Universal Robots URScript: Main Program plate.script

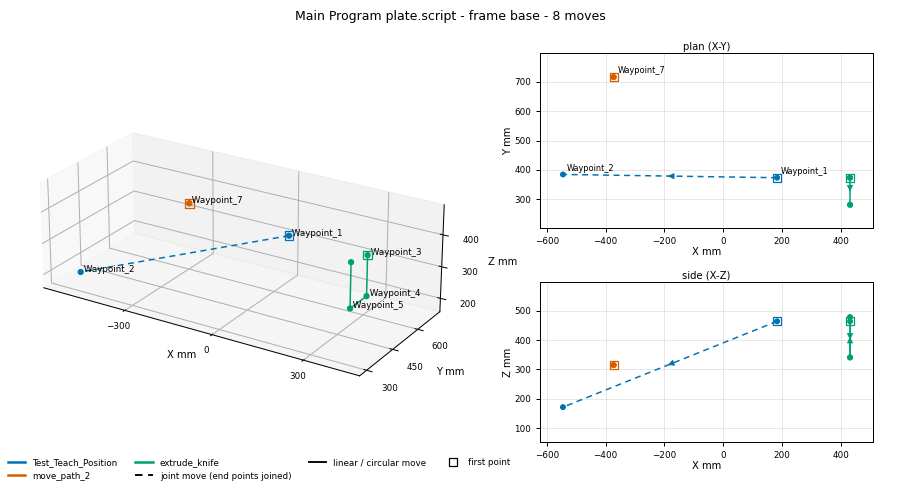
[picture p0: tool path of Main Program plate.script in frame base, 8 of 46 moves have a stored position in this frame; points joined in program order, loops and branches not executed]
def Main_Program_plate():
  global _hidden_verificationVariable=0
  set_gravity([0.0, 0.0, 9.82])
  set_tool_communication(False, 115200, 0, 1, 1.5, 3.5)
  set_tool_output_mode(0)
  set_tool_digital_output_mode(0, 1)
  set_tool_digital_output_mode(1, 1)
  set_tool_voltage(0)
  set_standard_analog_input_domain(0, 1)
  set_standard_analog_input_domain(1, 1)
  set_tool_analog_input_domain(0, 1)
  set_tool_analog_input_domain(1, 1)
  set_analog_outputdomain(0, 0)
  set_analog_outputdomain(1, 0)
  set_input_actions_to_default()
  set_target_payload(2.760000, [0.004000, -0.022000, 0.072000], [0.008360, 0.008360, 0.008360, 0.000000, 0.000000, 0.000000])
  set_safety_mode_transition_hardness(1)
  set_tcp(p[0.00855,-0.26517,0.10876999999999999,1.2092,-1.2092,1.2092])
  global Point_1=p[0.0,0.0,0.0,0.0,0.0,0.0]
  # begin: URCap Installation Node
  #   Source: MachineLogic for Universal Robots, 3.1.7, Vention Inc.
  #   Type: MachineLogic for Universal Robots
  def waitForResponse(expected_response_vention, cname_vention):
  response_vention = socket_read_string(cname_vention,timeout=15)
  while response_vention != expected_response_vention:
  sleep(0.01)
  response_vention = socket_read_string(cname_vention,timeout=15)
  end
  sleep(0.01)
  sync()
  end
  def sendString(string_vention, expected_response_vention, cname_vention):
  socket_send_string(str_cat(string_vention,";"), cname_vention)
  response_vention = socket_read_string(cname_vention,timeout=15)
  if(response_vention == "nAck"):
  popup("nAck received")
  end
  while response_vention != expected_response_vention:
  sleep(0.01)
  response_vention = socket_read_string(cname_vention,timeout=15)
  if(response_vention == "nAck"):
  popup("nAck received")
  end
  end
  sleep(0.01)
  sync()
  end
  def sendStringNAck(string_vention, expected_response_vention, cname_vention):
  socket_send_string(str_cat(string_vention,";"), cname_vention)
  response_vention = socket_read_string(cname_vention,timeout=15)
  if(response_vention == "nAck"):
  popup("nAck received")
  end
  while(response_vention != expected_response_vention and response_vention != "nAck"):
  sleep(0.01)
  response_vention = socket_read_string(cname_vention,timeout=15)
  if(response_vention == "nAck"):
  popup("nAck received",blocking=True)
  end
  end
  sleep(0.01)
  sync()
  end
  def sendStringWithTimeout(string_vention, expected_response_vention, cname_vention):
  socket_send_string(str_cat(string_vention,";"), cname_vention)
  response_vention = socket_read_string(cname_vention,timeout=10)
  if(response_vention == "nAck"):
  popup("nAck received"+string_vention)
  end
  sleep(0.01)
  sync()
  end
  def pollString(string_vention, expected_response_vention, cname_vention):
  socket_send_string(str_cat(string_vention,";"), cname_vention)
  response_vention = socket_read_string(cname_vention,timeout=15)
  if(response_vention == "nAck"):
  popup("nAck received")
  end
  while response_vention != expected_response_vention:
  sleep(1)
  socket_send_string(str_cat(string_vention,";"), cname_vention)
  response_vention = socket_read_string(cname_vention,timeout=15)
  if(response_vention == "nAck"):
  popup("nAck received")
  end
  end
  sleep(0.01)
  sync()
  end
  def sendVariable(var_vention, data_vention, expected_response_vention, cname_vention):
  socket_set_var(var_vention, data_vention, cname_vention)
  response_vention = socket_read_string(cname_vention,timeout=15)
  if(response_vention == "nAck"):
  popup("nAck received")
  end
  while response_vention != expected_response_vention:
  sleep(0.01)
  response_vention = socket_read_string(cname_vention,timeout=15)
  if(response_vention == "nAck"):
  popup("nAck received")
  end
  end
  sleep(0.01)
  sync()
  end
  def intToString(integer_vention,cname_vention):
  stringFix=""
  multiplier_vention123=1
  if integer_vention<0:
  stringFix="-"
  multiplier_vention123=-1
  end
  socket_set_var("GetString",integer_vention*multiplier_vention123,cname_vention)
  string_vention=""
  while string_vention=="":
  sleep(0.01)
  string_vention=socket_read_string(cname_vention,timeout=15)
  end
  sleep(0.01)
  sync()
  string_vention=stringFix+string_vention
  return string_vention
  end
  string_vention=""
  isVentionMovementBusy = False
  isVentionParallelMovementSendingScript = False
  ventionThreadHandle = 1
  isVentionMovementBusyMachineMotion1 = False
  isVentionParallelMovementSendingScriptMachineMotion1 = False
  socket_vention = socket_open("192.168.3.52", 9999, "MachineMotion1")
  if socket_vention==False:
  popup("Check configuration, can't connect to MachineMotion")
  end
  waitForResponse("MachineMotion connection established", "MachineMotion1")
  sendString("isReady", "MachineMotion isReady = true", "MachineMotion1")
  sendStringWithTimeout("setURCapVersion2", "setURCapVersion loaded", "MachineMotion1")
  sendString("SET speed_v2 1000000", "Ack", "MachineMotion1")
  sendString("SET acceleration_v2 100000", "Ack", "MachineMotion1")
  sendString("SET de_axis_1_microsteps_config 8", "Ack", "MachineMotion1")
  sendString("SET de_axis_1_mechanical_gain_config_v2 150000.0", "Ack", "MachineMotion1")
  sendString("SET de_axis_1_direction_config 1", "Ack", "MachineMotion1")
  sendString("SET de_axis_1_type_config Custom Actuator ", "Ack", "MachineMotion1")
  sendString("de_axis_1_config_exec", "Ack", "MachineMotion1")
  # end: URCap Installation Node
  step_count_0051c65f_c852_4209_9f2c_4b505770215d = 0.0
  thread Step_Counter_Thread_5b8e0ddc_5ea6_4297_b154_0c0ef5e6be23():
    while (True):
      step_count_0051c65f_c852_4209_9f2c_4b505770215d = step_count_0051c65f_c852_4209_9f2c_4b505770215d + 1.0
      sync()
    end
  end
  run Step_Counter_Thread_5b8e0ddc_5ea6_4297_b154_0c0ef5e6be23()
  global freedrive_m_var=  False
  global Waypoint_1_p=p[.183612702909, .373491415748, .464002429884, -.000031211095, 3.141572859461, .000004622808]
  global Waypoint_1_q=[-2.527531687413351, -2.1028810940184535, 2.591139856969015, -2.0582763157286585, -1.5713656584369105, 2.1834325790405273]
  global Waypoint_2_p=p[-.545552386461, .384638463642, .171639485768, .668511604681, -1.949272130073, 1.726627182696]
  global Waypoint_2_q=[-1.0565226713763636, -1.0868892234614869, 2.1878750959979456, -1.2335426074317475, -1.0471814314471644, 2.53226637840271]
  global Waypoint_7_p=p[-.372860657265, .716170383118, .314676530127, 1.570809017190, -.000000152759, .000003968716]
  global Waypoint_7_q=[-1.3816140333758753, -1.0546258252910157, 1.8334205786334437, -0.7777959269336243, -1.3827489058123987, 6.28196907043457]
  global Waypoint_8_p=p[-.372860657265, .716170383118, .314676530127, 1.570809017190, -.000000152759, .000003968716]
  global Waypoint_8_q=[-1.3816140333758753, -1.0546258252910157, 1.8334205786334437, -0.7777959269336243, -1.3827489058123987, 6.28196907043457]
  def calculate_point_to_move_towards(feature, direction, position_distance):
    local posDir=[direction[0], direction[1], direction[2]]
    if (norm(posDir) < 1e-6):
      return get_target_waypoint()
    end
    local direction_vector_normalized=normalize(posDir)
    local displacement_pose=p[direction_vector_normalized[0] * position_distance,direction_vector_normalized[1] * position_distance,direction_vector_normalized[2] * position_distance,0,0,0]
    local wanted_displacement_in_base_frame=pose_sub(pose_trans(feature, displacement_pose), feature)
    return pose_add(get_target_waypoint(), wanted_displacement_in_base_frame)
  end
  global Waypoint_3_p=p[.432120633847, .373496143704, .463992564600, -.000014136521, -3.141567738104, -.000014867905]
  global Waypoint_3_q=[-2.7853482405291956, -1.8143698177733363, 2.4549508730517786, -2.210560461083883, -1.5711315313922327, 1.9254603385925293]
  global Waypoint_4_p=p[.432136735069, .373501596410, .340883510249, -.000031606225, -3.141589553529, -.000013823620]
  global Waypoint_4_q=[-2.785483185444967, -1.6431261501707972, 2.568024222050802, -2.49489750484609, -1.5709694067584437, 1.9253177642822266]
  global Waypoint_5_p=p[.432160287104, .281352183882, .340893061994, .000015375091, 3.141574034920, .000032661568]
  global Waypoint_5_q=[-2.9616554419146937, -1.7250400982298792, 2.631975237523214, -2.4769565067686976, -1.5710294882403772, 1.7491776943206787]
  global Waypoint_6_p=p[.432128063058, .281346135716, .478493221894, .000013346378, -3.141574975494, -.000002942308]
  global Waypoint_6_q=[-2.961463991795675, -1.9219290218748988, 2.4929660002337855, -2.141019483605856, -1.571230713521139, 1.7493857145309448]
  def Test_Teach_Position():
    $ 9 "Test_Teach_Position" "noBreak"
    $ 10 "Home"
    movej([3.914755602117965, -2.1714491197731522, 2.311394911862933, -0.1410643170171042, 2.343248137569991, -7.705511093680784E-4], a=1.3962634015954636, v=1.0471975511965976)
    $ 11 "MoveL"
    $ 12 "Waypoint_1" "breakAfter"
    movel(Waypoint_1_p, a=1.2, v=0.25)
    $ 13 "'move welder up out of holder'"
    # 'move welder up out of holder'
    $ 14 "MoveJ"
    $ 15 "Waypoint_2" "breakAfter"
    movej(get_inverse_kin(Waypoint_2_p, qnear=Waypoint_2_q), a=1.3962634015954636, v=1.0471975511965976)
    $ 16 "freedrive_m_var≔ False "
    global freedrive_m_var=  False
    $ 17 "freedrive_m_var≔ True "
    global freedrive_m_var=  True
    $ 18 "Popup: Move the robot to the peg center, then click 'Continue'"
    popup("Move the robot to the peg center, then click 'Continue'", "Message", False, False, blocking=True)
    $ 19 "freedrive_m_var≔ False "
    global freedrive_m_var=  False
    $ 20 "Wait: 0.25"
    sleep(0.25)
    $ 21 "sync()"
    sync()
    $ 22 "tcp_pose≔get_actual_joint_positions()"
    global tcp_pose= get_actual_joint_positions ()
  end
  def move_path_2():
    $ 23 "move_path_2" "noBreak"
    $ 24 "pa1≔path1[1]"
    global pa1=path1[1]
    $ 25 "pa2≔path1[2]"
    global pa2=path1[2]
    $ 26 "p1≔path1[3]"
    global p1=path1[3]
    $ 27 "p2≔path1[4]"
    global p2=path1[4]
    $ 28 "p3≔path1[5]"
    global p3=path1[5]
    $ 29 "p4≔path1[6]"
    global p4=path1[6]
    $ 30 "p5≔path1[7]"
    global p5=path1[7]
    $ 31 "pr1≔path1[8]"
    global pr1=path1[8]
    $ 32 "MoveJ"
    $ 33 "Waypoint_7" "breakAfter"
    movej(get_inverse_kin(Waypoint_7_p, qnear=Waypoint_7_q), a=1.3962634015954636, v=1.0471975511965976)
    $ 34 "MoveJ"
    $ 35 "pa1" "breakAfter"
    movej(pa1, a=1.3962634015954636, v=1.0471975511965976)
    $ 36 "MoveL"
    $ 37 "pa2" "breakAfter"
    movel(pa2, a=1.2, v=0.2)
    $ 38 "MoveL"
    $ 39 "p1" "breakAfter"
    movel(p1, a=1.2, v=0.05)
    $ 40 "Wait: 1.0"
    sleep(1.0)
    $ 41 "MoveL"
    $ 42 "p2" "breakAfter"
    movel(p2, a=1.2, v=0.012)
    $ 43 "MoveP"
    $ 44 "CircleMove"
    $ 45 "p3" "noBreak"
    $ 46 "p4" "breakAfter"
    movec(p3, p4, a=1.2, v=5.0E-4, r=0.0, mode=1)
    $ 47 "MoveL"
    $ 48 "p5" "breakAfter"
    movel(p5, a=1.2, v=0.012)
    $ 49 "MoveL"
    $ 50 "pr1" "breakAfter"
    movel(pr1, a=1.2, v=0.25)
    $ 51 "MoveJ"
    $ 52 "Waypoint_8" "breakAfter"
    movej(get_inverse_kin(Waypoint_8_p, qnear=Waypoint_8_q), a=1.3962634015954636, v=1.0471975511965976)
  end
  def Corner_Homing_BRB():
    $ 53 "Corner_Homing_BRB" "noBreak"
    $ 54 "'Use this program when tool is already positioned close to corner (back right bottom corner)'"
    # 'Use this program when tool is already positioned close to corner (back right bottom corner)'
    $ 55 "'tool flange will seek all 3 sides. will save those 5 locs in p__'"
    # 'tool flange will seek all 3 sides. will save those 5 locs in p__'
    $ 56 "align_tcp_left()"
    align_tcp_left()
    $ 57 "'right side'"
    # 'right side'
    $ 58 "MoveL"
    $ 59 "Direction: Base X-"
    global move_thread_flag_59=0
    thread move_thread_59():
      enter_critical
      move_thread_flag_59 = 1
      local towardsPos=calculate_point_to_move_towards(p[0.0,0.0,0.0,0.0,0.0,0.0], [-1.0,0.0,0.0], 0.05)
      movel(towardsPos, a=1.2, v=0.25)
      move_thread_flag_59 = 2
      exit_critical
    end
    move_thread_flag_59 = 0
    move_thread_han_59 = run move_thread_59()
    while (True):
      sleep(1.0E-10)
      if (move_thread_flag_59 > 1):
        join move_thread_han_59
        $ 60 "Until (distance)"
        break
      end
      sync()
    end
    $ 61 "MoveL"
    $ 62 "Direction: Base Y-"
    global move_thread_flag_62=0
    thread move_thread_62():
      enter_critical
      move_thread_flag_62 = 1
      local towardsPos=calculate_point_to_move_towards(p[0.0,0.0,0.0,0.0,0.0,0.0], [0.0,-1.0,0.0], 1000.0)
      movel(towardsPos, a=1.2, v=0.05)
      move_thread_flag_62 = 2
      exit_critical
    end
    move_thread_flag_62 = 0
    move_thread_han_62 = run move_thread_62()
    while (True):
      local targetTcpDirection=get_target_tcp_speed()
      local stepsToRetract=tool_contact(direction=targetTcpDirection)
      if (stepsToRetract > 0):
        kill move_thread_han_62
        stopl(3.0)
        local backTrackMovement=get_actual_joint_positions_history(stepsToRetract)
        local contactPose=get_forward_kin(backTrackMovement)
        local posDir=[targetTcpDirection[0],targetTcpDirection[1],targetTcpDirection[2]]
        local retractTo=contactPose
        if (norm(posDir) > 1e-6):
          local normalizedPosDir=normalize(posDir)
          local additionalRetraction=p[normalizedPosDir[0] * 0.0, normalizedPosDir[1] * 0.0, normalizedPosDir[2] * 0.0, 0, 0, 0]
          retractTo = pose_sub(contactPose, additionalRetraction)
        end
        movel(retractTo, a=3.0, v=0.1)
        $ 63 "Until (tool_contact_detection)"
        break
      end
      sync()
    end
    $ 64 "p11≔get_actual_tcp_pose()"
    global p11= get_actual_tcp_pose ()
    $ 65 "MoveL"
    $ 66 "Direction: Base Y+"
    global move_thread_flag_66=0
    thread move_thread_66():
      enter_critical
      move_thread_flag_66 = 1
      local towardsPos=calculate_point_to_move_towards(p[0.0,0.0,0.0,0.0,0.0,0.0], [0.0,1.0,0.0], 0.05)
      movel(towardsPos, a=1.2, v=0.25)
      move_thread_flag_66 = 2
      exit_critical
    end
    move_thread_flag_66 = 0
    move_thread_han_66 = run move_thread_66()
    while (True):
      sleep(1.0E-10)
      if (move_thread_flag_66 > 1):
        join move_thread_han_66
        $ 67 "Until (distance)"
        break
      end
      sync()
    end
    $ 68 "MoveL"
    $ 69 "Direction: Base X-"
    global move_thread_flag_69=0
    thread move_thread_69():
      enter_critical
      move_thread_flag_69 = 1
      local towardsPos=calculate_point_to_move_towards(p[0.0,0.0,0.0,0.0,0.0,0.0], [-1.0,0.0,0.0], 0.15)
      movel(towardsPos, a=1.2, v=0.25)
      move_thread_flag_69 = 2
      exit_critical
    end
    move_thread_flag_69 = 0
    move_thread_han_69 = run move_thread_69()
    while (True):
      sleep(1.0E-10)
      if (move_thread_flag_69 > 1):
        join move_thread_han_69
        $ 70 "Until (distance)"
        break
      end
      sync()
    end
    $ 71 "MoveL"
    $ 72 "Direction: Base Y-"
    global move_thread_flag_72=0
    thread move_thread_72():
      enter_critical
      move_thread_flag_72 = 1
      local towardsPos=calculate_point_to_move_towards(p[0.0,0.0,0.0,0.0,0.0,0.0], [0.0,-1.0,0.0], 1000.0)
      movel(towardsPos, a=1.2, v=0.05)
      move_thread_flag_72 = 2
      exit_critical
    end
    move_thread_flag_72 = 0
    move_thread_han_72 = run move_thread_72()
    while (True):
      local targetTcpDirection=get_target_tcp_speed()
      local stepsToRetract=tool_contact(direction=targetTcpDirection)
      if (stepsToRetract > 0):
        kill move_thread_han_72
        stopl(3.0)
        local backTrackMovement=get_actual_joint_positions_history(stepsToRetract)
        local contactPose=get_forward_kin(backTrackMovement)
        local posDir=[targetTcpDirection[0],targetTcpDirection[1],targetTcpDirection[2]]
        local retractTo=contactPose
        if (norm(posDir) > 1e-6):
          local normalizedPosDir=normalize(posDir)
          local additionalRetraction=p[normalizedPosDir[0] * 0.0, normalizedPosDir[1] * 0.0, normalizedPosDir[2] * 0.0, 0, 0, 0]
          retractTo = pose_sub(contactPose, additionalRetraction)
        end
        movel(retractTo, a=3.0, v=0.1)
        $ 73 "Until (tool_contact_detection)"
        break
      end
      sync()
    end
    $ 74 "p12≔get_actual_tcp_pose()"
    global p12= get_actual_tcp_pose ()
    $ 75 "MoveL"
    $ 76 "Direction: Base Y+"
    global move_thread_flag_76=0
    thread move_thread_76():
      enter_critical
      move_thread_flag_76 = 1
      local towardsPos=calculate_point_to_move_towards(p[0.0,0.0,0.0,0.0,0.0,0.0], [0.0,1.0,0.0], 0.05)
      movel(towardsPos, a=1.2, v=0.25)
      move_thread_flag_76 = 2
      exit_critical
    end
    move_thread_flag_76 = 0
    move_thread_han_76 = run move_thread_76()
    while (True):
      sleep(1.0E-10)
      if (move_thread_flag_76 > 1):
        join move_thread_han_76
        $ 77 "Until (distance)"
        break
      end
      sync()
    end
    $ 78 "MoveL"
    $ 79 "Direction: Base X+"
    global move_thread_flag_79=0
    thread move_thread_79():
      enter_critical
      move_thread_flag_79 = 1
      local towardsPos=calculate_point_to_move_towards(p[0.0,0.0,0.0,0.0,0.0,0.0], [1.0,0.0,0.0], 0.3)
      movel(towardsPos, a=1.2, v=0.25)
      move_thread_flag_79 = 2
      exit_critical
    end
    move_thread_flag_79 = 0
    move_thread_han_79 = run move_thread_79()
    while (True):
      sleep(1.0E-10)
      if (move_thread_flag_79 > 1):
        join move_thread_han_79
        $ 80 "Until (distance)"
        break
      end
      sync()
    end
    $ 81 "align_tcp_forward()"
    align_tcp_forward()
    $ 82 "'back side'"
    # 'back side'
    $ 83 "MoveL"
    $ 84 "Direction: Base Y-"
    global move_thread_flag_84=0
    thread move_thread_84():
      enter_critical
      move_thread_flag_84 = 1
      local towardsPos=calculate_point_to_move_towards(p[0.0,0.0,0.0,0.0,0.0,0.0], [0.0,-1.0,0.0], 0.1)
      movel(towardsPos, a=1.2, v=0.25)
      move_thread_flag_84 = 2
      exit_critical
    end
    move_thread_flag_84 = 0
    move_thread_han_84 = run move_thread_84()
    while (True):
      sleep(1.0E-10)
      if (move_thread_flag_84 > 1):
        join move_thread_han_84
        $ 85 "Until (distance)"
        break
      end
      sync()
    end
    $ 86 "MoveL"
    $ 87 "Direction: Base X-"
    global move_thread_flag_87=0
    thread move_thread_87():
      enter_critical
      move_thread_flag_87 = 1
      local towardsPos=calculate_point_to_move_towards(p[0.0,0.0,0.0,0.0,0.0,0.0], [-1.0,0.0,0.0], 1000.0)
      movel(towardsPos, a=1.2, v=0.05)
      move_thread_flag_87 = 2
      exit_critical
    end
    move_thread_flag_87 = 0
    move_thread_han_87 = run move_thread_87()
    while (True):
      local targetTcpDirection=get_target_tcp_speed()
      local stepsToRetract=tool_contact(direction=targetTcpDirection)
      if (stepsToRetract > 0):
        kill move_thread_han_87
        stopl(3.0)
        local backTrackMovement=get_actual_joint_positions_history(stepsToRetract)
        local contactPose=get_forward_kin(backTrackMovement)
        local posDir=[targetTcpDirection[0],targetTcpDirection[1],targetTcpDirection[2]]
        local retractTo=contactPose
        if (norm(posDir) > 1e-6):
          local normalizedPosDir=normalize(posDir)
          local additionalRetraction=p[normalizedPosDir[0] * 0.0, normalizedPosDir[1] * 0.0, normalizedPosDir[2] * 0.0, 0, 0, 0]
          retractTo = pose_sub(contactPose, additionalRetraction)
        end
        movel(retractTo, a=3.0, v=0.1)
        $ 88 "Until (tool_contact_detection)"
        break
      end
      sync()
    end
    $ 89 "p21≔get_actual_tcp_pose()"
    global p21= get_actual_tcp_pose ()
    $ 90 "MoveL"
    $ 91 "Direction: Base X+"
    global move_thread_flag_91=0
    thread move_thread_91():
      enter_critical
      move_thread_flag_91 = 1
      local towardsPos=calculate_point_to_move_towards(p[0.0,0.0,0.0,0.0,0.0,0.0], [1.0,0.0,0.0], 0.05)
      movel(towardsPos, a=1.2, v=0.25)
      move_thread_flag_91 = 2
      exit_critical
    end
    move_thread_flag_91 = 0
    move_thread_han_91 = run move_thread_91()
    while (True):
      sleep(1.0E-10)
      if (move_thread_flag_91 > 1):
        join move_thread_han_91
        $ 92 "Until (distance)"
        break
      end
      sync()
    end
    $ 93 "MoveL"
    $ 94 "Direction: Base Y-"
    global move_thread_flag_94=0
    thread move_thread_94():
      enter_critical
      move_thread_flag_94 = 1
      local towardsPos=calculate_point_to_move_towards(p[0.0,0.0,0.0,0.0,0.0,0.0], [0.0,-1.0,0.0], 0.15)
      movel(towardsPos, a=1.2, v=0.25)
      move_thread_flag_94 = 2
      exit_critical
    end
    move_thread_flag_94 = 0
    move_thread_han_94 = run move_thread_94()
    while (True):
      sleep(1.0E-10)
      if (move_thread_flag_94 > 1):
        join move_thread_han_94
        $ 95 "Until (distance)"
        break
      end
      sync()
    end
    $ 96 "MoveL"
    $ 97 "Direction: Base X-"
    global move_thread_flag_97=0
    thread move_thread_97():
      enter_critical
      move_thread_flag_97 = 1
      local towardsPos=calculate_point_to_move_towards(p[0.0,0.0,0.0,0.0,0.0,0.0], [-1.0,0.0,0.0], 1000.0)
      movel(towardsPos, a=1.2, v=0.05)
      move_thread_flag_97 = 2
      exit_critical
    end
    move_thread_flag_97 = 0
    move_thread_han_97 = run move_thread_97()
    while (True):
      local targetTcpDirection=get_target_tcp_speed()
      local stepsToRetract=tool_contact(direction=targetTcpDirection)
      if (stepsToRetract > 0):
        kill move_thread_han_97
        stopl(3.0)
        local backTrackMovement=get_actual_joint_positions_history(stepsToRetract)
        local contactPose=get_forward_kin(backTrackMovement)
        local posDir=[targetTcpDirection[0],targetTcpDirection[1],targetTcpDirection[2]]
        local retractTo=contactPose
        if (norm(posDir) > 1e-6):
          local normalizedPosDir=normalize(posDir)
          local additionalRetraction=p[normalizedPosDir[0] * 0.0, normalizedPosDir[1] * 0.0, normalizedPosDir[2] * 0.0, 0, 0, 0]
          retractTo = pose_sub(contactPose, additionalRetraction)
        end
        movel(retractTo, a=3.0, v=0.1)
        $ 98 "Until (tool_contact_detection)"
        break
      end
      sync()
    end
    $ 99 "p22≔get_actual_tcp_pose()"
    global p22= get_actual_tcp_pose ()
    $ 100 "MoveL"
    $ 101 "Direction: Base X+"
    global move_thread_flag_101=0
    thread move_thread_101():
      enter_critical
      move_thread_flag_101 = 1
      local towardsPos=calculate_point_to_move_towards(p[0.0,0.0,0.0,0.0,0.0,0.0], [1.0,0.0,0.0], 0.05)
      movel(towardsPos, a=1.2, v=0.25)
      move_thread_flag_101 = 2
      exit_critical
    end
    move_thread_flag_101 = 0
    move_thread_han_101 = run move_thread_101()
    while (True):
      sleep(1.0E-10)
      if (move_thread_flag_101 > 1):
        join move_thread_han_101
        $ 102 "Until (distance)"
        break
      end
      sync()
    end
    $ 103 "'regroup for up turn'"
    # 'regroup for up turn'
    $ 104 "MoveL"
    $ 105 "Direction: Base X+"
    global move_thread_flag_105=0
    thread move_thread_105():
      enter_critical
      move_thread_flag_105 = 1
      local towardsPos=calculate_point_to_move_towards(p[0.0,0.0,0.0,0.0,0.0,0.0], [1.0,0.0,0.0], 0.2)
      movel(towardsPos, a=1.2, v=0.25)
      move_thread_flag_105 = 2
      exit_critical
    end
    move_thread_flag_105 = 0
    move_thread_han_105 = run move_thread_105()
    while (True):
      sleep(1.0E-10)
      if (move_thread_flag_105 > 1):
        join move_thread_han_105
        $ 106 "Until (distance)"
        break
      end
      sync()
    end
    $ 107 "Direction: Base Y+"
    global move_thread_flag_107=0
    thread move_thread_107():
      enter_critical
      move_thread_flag_107 = 1
      local towardsPos=calculate_point_to_move_towards(p[0.0,0.0,0.0,0.0,0.0,0.0], [0.0,1.0,0.0], 0.5)
      movel(towardsPos, a=1.2, v=0.25)
      move_thread_flag_107 = 2
      exit_critical
    end
    move_thread_flag_107 = 0
    move_thread_han_107 = run move_thread_107()
    while (True):
      sleep(1.0E-10)
      if (move_thread_flag_107 > 1):
        join move_thread_han_107
        $ 108 "Until (distance)"
        break
      end
      sync()
    end
    $ 109 "MoveL"
    $ 110 "Direction: Base Z-"
    global move_thread_flag_110=0
    thread move_thread_110():
      enter_critical
      move_thread_flag_110 = 1
      local towardsPos=calculate_point_to_move_towards(p[0.0,0.0,0.0,0.0,0.0,0.0], [0.0,0.0,-1.0], 0.1)
      movel(towardsPos, a=1.2, v=0.25)
      move_thread_flag_110 = 2
      exit_critical
    end
    move_thread_flag_110 = 0
    move_thread_han_110 = run move_thread_110()
    while (True):
      sleep(1.0E-10)
      if (move_thread_flag_110 > 1):
        join move_thread_han_110
        $ 111 "Until (distance)"
        break
      end
      sync()
    end
    $ 112 "align_tcp_up()"
    align_tcp_up()
    $ 113 "MoveL"
    $ 114 "Direction: Base X-"
    global move_thread_flag_114=0
    thread move_thread_114():
      enter_critical
      move_thread_flag_114 = 1
      local towardsPos=calculate_point_to_move_towards(p[0.0,0.0,0.0,0.0,0.0,0.0], [-1.0,0.0,0.0], 0.25)
      movel(towardsPos, a=1.2, v=0.25)
      move_thread_flag_114 = 2
      exit_critical
    end
    move_thread_flag_114 = 0
    move_thread_han_114 = run move_thread_114()
    while (True):
      sleep(1.0E-10)
      if (move_thread_flag_114 > 1):
        join move_thread_han_114
        $ 115 "Until (distance)"
        break
      end
      sync()
    end
    $ 116 "Direction: Base Y-"
    global move_thread_flag_116=0
    thread move_thread_116():
      enter_critical
      move_thread_flag_116 = 1
      local towardsPos=calculate_point_to_move_towards(p[0.0,0.0,0.0,0.0,0.0,0.0], [0.0,-1.0,0.0], 0.32)
      movel(towardsPos, a=1.2, v=0.25)
      move_thread_flag_116 = 2
      exit_critical
    end
    move_thread_flag_116 = 0
    move_thread_han_116 = run move_thread_116()
    while (True):
      sleep(1.0E-10)
      if (move_thread_flag_116 > 1):
        join move_thread_han_116
        $ 117 "Until (distance)"
        break
      end
      sync()
    end
    $ 118 "'bottom side'"
    # 'bottom side'
    $ 119 "MoveL"
    $ 120 "Direction: Base Z+"
    global move_thread_flag_120=0
    thread move_thread_120():
      enter_critical
      move_thread_flag_120 = 1
      local towardsPos=calculate_point_to_move_towards(p[0.0,0.0,0.0,0.0,0.0,0.0], [0.0,0.0,1.0], 1000.0)
      movel(towardsPos, a=1.2, v=0.05)
      move_thread_flag_120 = 2
      exit_critical
    end
    move_thread_flag_120 = 0
    move_thread_han_120 = run move_thread_120()
    while (True):
      local targetTcpDirection=get_target_tcp_speed()
      local stepsToRetract=tool_contact(direction=targetTcpDirection)
      if (stepsToRetract > 0):
        kill move_thread_han_120
        stopl(3.0)
        local backTrackMovement=get_actual_joint_positions_history(stepsToRetract)
        local contactPose=get_forward_kin(backTrackMovement)
        local posDir=[targetTcpDirection[0],targetTcpDirection[1],targetTcpDirection[2]]
        local retractTo=contactPose
        if (norm(posDir) > 1e-6):
          local normalizedPosDir=normalize(posDir)
          local additionalRetraction=p[normalizedPosDir[0] * 0.0, normalizedPosDir[1] * 0.0, normalizedPosDir[2] * 0.0, 0, 0, 0]
          retractTo = pose_sub(contactPose, additionalRetraction)
        end
        movel(retractTo, a=3.0, v=0.1)
        $ 121 "Until (tool_contact_detection)"
        break
      end
      sync()
    end
    $ 122 "p3≔get_actual_tcp_pose()"
    global p3= get_actual_tcp_pose ()
    $ 123 "MoveL"
    $ 124 "Direction: Base Z-"
    global move_thread_flag_124=0
    thread move_thread_124():
      enter_critical
      move_thread_flag_124 = 1
      local towardsPos=calculate_point_to_move_towards(p[0.0,0.0,0.0,0.0,0.0,0.0], [0.0,0.0,-1.0], 0.05)
      movel(towardsPos, a=1.2, v=0.25)
      move_thread_flag_124 = 2
      exit_critical
    end
    move_thread_flag_124 = 0
    move_thread_han_124 = run move_thread_124()
    while (True):
      sleep(1.0E-10)
      if (move_thread_flag_124 > 1):
        join move_thread_han_124
        $ 125 "Until (distance)"
        break
      end
      sync()
    end
    $ 126 "MoveL"
    $ 127 "Direction: Base X+"
    global move_thread_flag_127=0
    thread move_thread_127():
      enter_critical
      move_thread_flag_127 = 1
      local towardsPos=calculate_point_to_move_towards(p[0.0,0.0,0.0,0.0,0.0,0.0], [1.0,0.0,0.0], 0.1)
      movel(towardsPos, a=1.2, v=0.25)
      move_thread_flag_127 = 2
      exit_critical
    end
    move_thread_flag_127 = 0
    move_thread_han_127 = run move_thread_127()
    while (True):
      sleep(1.0E-10)
      if (move_thread_flag_127 > 1):
        join move_thread_han_127
        $ 128 "Until (distance)"
        break
      end
      sync()
    end
    $ 129 "Direction: Base Y+"
    global move_thread_flag_129=0
    thread move_thread_129():
      enter_critical
      move_thread_flag_129 = 1
      local towardsPos=calculate_point_to_move_towards(p[0.0,0.0,0.0,0.0,0.0,0.0], [0.0,1.0,0.0], 0.1)
      movel(towardsPos, a=1.2, v=0.25)
      move_thread_flag_129 = 2
      exit_critical
    end
    move_thread_flag_129 = 0
    move_thread_han_129 = run move_thread_129()
    while (True):
      sleep(1.0E-10)
      if (move_thread_flag_129 > 1):
        join move_thread_han_129
        $ 130 "Until (distance)"
        break
      end
      sync()
    end
  end
  def extrude_knife():
    $ 131 "extrude_knife" "noBreak"
    $ 132 "'Move to bucket'"
    # 'Move to bucket'
    $ 133 "MoveJ"
    $ 134 "Waypoint_3" "breakAfter"
    movej(get_inverse_kin(Waypoint_3_p, qnear=Waypoint_3_q), a=1.3962634015954636, v=1.0471975511965976)
    $ 135 "MoveL"
    $ 136 "Waypoint_4" "breakAfter"
    movel(Waypoint_4_p, a=1.2, v=0.25)
    $ 137 "'extrude out a foot'"
    # 'extrude out a foot'
    $ 138 "Wait: 1.0"
    sleep(1.0)
    $ 139 "MoveL"
    $ 140 "'slice over knife'"
    # 'slice over knife'
    $ 141 "Waypoint_5" "breakAfter"
    movel(Waypoint_5_p, a=1.2, v=0.04)
    $ 142 "MoveL"
    $ 143 "Waypoint_6" "breakAfter"
    movel(Waypoint_6_p, a=1.2, v=0.25)
    $ 144 "'raise up away from knife'"
    # 'raise up away from knife'
  end
  def align_tcp_left():
    $ 145 "align_tcp_left" "noBreak"
    $ 146 "'this program aligns the tcp parallel to the y direction'"
    # 'this program aligns the tcp parallel to the y direction'
    $ 147 "cp≔get_actual_tcp_pose()"
    global cp= get_actual_tcp_pose ()
    $ 148 "aligned_y_pose≔p[cp[0],cp[1],cp[2],1.570796,0,0]"
    global aligned_y_pose=p[cp[0],cp[1],cp[2],1.570796,0,0]
    $ 149 "MoveJ"
    $ 150 "aligned_y_pose" "breakAfter"
    movej(aligned_y_pose, a=1.3962634015954636, v=1.0471975511965976)
  end
  def align_tcp_up():
    $ 151 "align_tcp_up" "noBreak"
    $ 152 "'this program aligns the tcp parallel to the y direction'"
    # 'this program aligns the tcp parallel to the y direction'
    $ 153 "cp≔get_actual_tcp_pose()"
    global cp= get_actual_tcp_pose ()
    $ 154 "aligned_y_pose≔p[cp[0],cp[1],cp[2],0,0,0]"
    global aligned_y_pose=p[cp[0],cp[1],cp[2],0,0,0]
    $ 155 "MoveJ"
    $ 156 "aligned_y_pose" "breakAfter"
    movej(aligned_y_pose, a=1.3962634015954636, v=1.0471975511965976)
  end
  def align_tcp_forward():
    $ 157 "align_tcp_forward" "noBreak"
    $ 158 "'this program aligns the tcp parallel to the y direction'"
    # 'this program aligns the tcp parallel to the y direction'
    $ 159 "cp≔get_actual_tcp_pose()"
    global cp= get_actual_tcp_pose ()
    $ 160 "aligned_y_pose≔p[cp[0],cp[1],cp[2],0,-1.570796,0]"
    global aligned_y_pose=p[cp[0],cp[1],cp[2],0,-1.570796,0]
    $ 161 "MoveJ"
    $ 162 "aligned_y_pose" "breakAfter"
    movej(aligned_y_pose, a=1.3962634015954636, v=1.0471975511965976)
  end
  $ 163 "Thread_1"
  thread Thread_1():
    while (True):
      $ 164 "Loop  True "
      while (  True  ):
        $ 165 "If freedrive_m_var≟ True "
        if (freedrive_m_var ==   True  ):
          $ 166 "freedrive_mode()"
          freedrive_mode()
        else:
          $ 167 "Else" "noBreak"
          $ 168 "end_freedrive_mode()"
          end_freedrive_mode()
        end
        $ 169 "sync()"
        sync()
      end
    end
  end
  threadId_Thread_1 = run Thread_1()
  $ 2 "Robot Program"
  $ 3 "Test_Teach_Position()"
  Test_Teach_Position()
  $ 4 "Corner_Homing_BRB()"
  Corner_Homing_BRB()
  $ 5 "extrude_knife()"
  extrude_knife()
  $ 6 "Script: analyze_touchpoints.script"
  # this file creates the function for analyzing touchpoints
  # define pi
  pi = 3.1415926535

  # it takes 5 arguments as points
  # it returns a struct containing: (pointintersect, pointapproach1, pointapproach2, point1, point2, point3, point4, point5, pointreturn1, heading1, heading2, heading3)
  def analyze_touchpoints(p11, p12, p21, p22, p3):
    # FIND THE INTERSECTION
    # comment get the z
    zcoord=p3[2]

    # get the raw points from the first line
    l1p1x=p11[0]
    l1p1y=p11[1]
    l1p2x=p12[0]
    l1p2y=p12[1]

    # equate the first line in 2d space
    ml1 = (l1p2y-l1p1y) / (l1p2x-l1p1x)

    # b = y - mx
    bl1 = l1p1y - ml1 * l1p1x

    # get the raw points from the second line
    l2p1x=p21[0]
    l2p1y=p21[1]
    l2p2x=p22[0]
    l2p2y=p22[1]

    # equate the second line in 2d space
    ml2 = (l2p2y-l2p1y) / (l2p2x-l2p1x)

    # b = y - mx
    bl2 = l2p1y - ml2 * l2p1x


    # find the intersection of the two lines
    # m1x+b1 = m2x+b2
    # m1x - m2x = b2 - b1
    # x = (b2-b1) / (m1-m2)
    xintersect = (bl2-bl1) / (ml1-ml2)
    yintersect = ml1 * xintersect + bl1

    #FIND THE VECTORS
    #define a vector from the intersection to the second point on the first line
    l1delxfull = l1p2x - xintersect
    l1delyfull = l1p2y - yintersect

    l1delmag = sqrt(l1delxfull*l1delxfull + l1delyfull*l1delyfull)

    l1delxunit = l1delxfull / l1delmag
    l1delyunit = l1delyfull / l1delmag

    #define a vector from the intersection to the second point on the second line
    l2delxfull = l2p2x - xintersect
    l2delyfull = l2p2y - yintersect

    l2delmag = sqrt(l2delxfull*l2delxfull + l2delyfull*l2delyfull)

    l2delxunit = l2delxfull / l2delmag
    l2delyunit = l2delyfull / l2delmag

    # FIND THE FOUR POINTS ON THE LINES
    # find locations 8 inches away from  intersect point
    # CONST
    welddistance = 8
    roundoverdistance = 0.05
    zup = .375
    # inches
    wd = welddistance * 25.4 / 1000
    rod = roundoverdistance * 25.4 / 1000
    zup = zup * 25.4 / 1000

    # now we have the unit vector. extend the weld distance from the intersection
    x = xintersect + l1delxunit * wd
    y = yintersect + l1delyunit * wd
    z = zcoord + zup

    point1 = p[x,y,z,1.570796,0,0] # dummy orientation for now

    x = xintersect + l1delxunit * rod
    y = yintersect + l1delyunit * rod

    point2 = p[x,y,z,1.570796,0,0]

    # now we have the unit vector. extend the weld distance from the intersection
    x = xintersect + l2delxunit * wd
    y = yintersect + l2delyunit * wd

    point5 = p[x,y,z,0,-1.570796,0]

    x = xintersect + l2delxunit * rod
    y = yintersect + l2delyunit * rod

    point4 = p[x,y,z,0,-1.570796,0]

    #DEFINE APPROACH POINTS
    pointintersect = p[xintersect,yintersect,zcoord,0,0,0]
    pointapproach1 = p[xintersect+0.1,yintersect+0.1,z,1.570796,0,0]
    pointapproach2 = p[point1[0], point1[1]+0.1, point1[2], point1[3], point1[4], point1[5]]
    pointreturn1 = p[point5[0]+0.1, point5[1], point5[2], point5[3], point5[4], point5[5]]

    #FIND HEADINGS
    #for each heading, find the angle of the line with respect to the pos x axis. then add/subtract 90 degrees because you want to be perpendicular to that
    headingvector1 = convert_uv_to_heading(l1delxunit, l1delyunit)
    headingvector2 = convert_uv_to_heading(l2delxunit, l2delyunit)
    # find halfway heading
    heading2 = (headingvector1 + headingvector2)/2
    # find headings that the robot should face while traveling, perpendicular to the vectors of the sides of the box
    heading1 = headingvector1 + pi/2
    heading3 = headingvector2 - pi/2

    #FIND POINT 3
    #see if we have to / can find point 3
    findpoint3 = True
    if roundoverdistance == 0:
      findpoint3 = False
    end
    if findpoint3:
      # i need to find the point3 such that the arc from p2 to p3 to p4 is tangent to p1-p2 and p4-p5. making this a smooth path will be good
      # the direction of movement is from pointintersect in the direction of heading2
      # how much movement though? this will depend on whether it is actually a 90 degree angle or not.
      # first, find the perpendicular lines through points 2 and 4
      perp2 = find_perpendicular_line(ml1, point2[0], point2[1])
      perp4 = find_perpendicular_line(ml2, point4[0], point4[1])
      # next, find the intersection of those two lines
      perpintersect = find_intersection(perp2[0], perp2[1], perp4[0], perp4[1])
      radiusofcircle = distance_between(perpintersect[0], perpintersect[1], 0, point2[0], point2[1], 0)
      # find a vector the direction of heading2
      uvx = cos(heading2)
      uvy = sin(heading2)
      # compute point3. pass in negative radius because the direction is into the tank but we want to move from the intersection out to the rounded edge.
      point3coords = add_vectordistance_to_point(perpintersect[0], perpintersect[1], z, uvx, uvy, 0, -1 * radiusofcircle)
      point3 = p[point3coords[0], point3coords[1], point3coords[2], 0, 0, 0]
    end

    #APPLY ACTUAL RXRYRZ TO POINTS
    # convert the headings to rxryrz and insert those values into the relevant points
    rxryrz = convert_heading_to_axang(heading1)
    rx = rxryrz[0]
    ry = rxryrz[1]
    rz = rxryrz[2]
    pointapproach1 = p[pointapproach1[0], pointapproach1[1], pointapproach1[2], rx, ry, rz]
    pointapproach2 = p[pointapproach2[0], pointapproach2[1], pointapproach2[2], rx, ry, rz]
    point1 = p[point1[0], point1[1], point1[2], rx, ry, rz]
    point2 = p[point2[0], point2[1], point2[2], rx, ry, rz]
    rxryrz = convert_heading_to_axang(heading2)
    rx = rxryrz[0]
    ry = rxryrz[1]
    rz = rxryrz[2]
    if findpoint3:
      point3 = p[point3[0], point3[1], point3[2], rx, ry, rz]
    else:
      point3 = point2
    end
    rxryrz = convert_heading_to_axang(heading3)
    rx = rxryrz[0]
    ry = rxryrz[1]
    rz = rxryrz[2]
    point4 = p[point4[0], point4[1], point4[2], rx, ry, rz]
    point5 = p[point5[0], point5[1], point5[2], rx, ry, rz]
    pointreturn1 = p[pointreturn1[0], pointreturn1[1], pointreturn1[2], rx, ry, rz]

    #RETURN STRUCT
    ret = struct(pointintersect=pointintersect, pointapproach1=pointapproach1, pointapproach2=pointapproach2, point1=point1, point2=point2, point3=point3, point4=point4, point5=point5, pointreturn1=pointreturn1, heading1=heading1, heading2=heading2, heading3=heading3)
    return ret
  end

  # this function converts a unit vector to its heading angle ccw from x+ axis
  # takes uvx and uvy
  # returns heading in radians
  def convert_uv_to_heading(uvx, uvy):
    baseang = atan(uvy/uvx)
    if uvx < 0:
      ang = baseang + pi
    elif uvy < 0:
      ang = baseang + pi * 2
    else:
      ang = baseang
    end
    return ang
  end

  # this function finds the equation of a line, perpendicular to a given line, and going through a given point
  # takes 3 arguments: m (the original line's slope), x (point's x coord), y (point's y coord). the b of the original line is not needed
  # returns a list of [m,b] (the slope and intercept of the new line)
  def find_perpendicular_line(origm, x, y):
    m = (1/origm) * -1
    b = y - m*x
    ret = [m, b]
    return ret
  end

  # this function finds the intersection point between two lines in the xy plane
  # takes 4 arguments: m1, b1, m2, b2
  # returns a list of [x,y] (the point of intersection)
  def find_intersection(m1, b1, m2, b2):
    # m1x+b1 = m2x+b2
    # m1x - m2x = b2 - b1
    # x = (b2-b1) / (m1-m2)
    x = (b2-b1) / (m1-m2)
    y = m1 * x + b1
    ret = [x, y]
    return ret
  end

  # this function finds the distance between 2 points in 3d space
  # it takes 6 arguments: x1, y1, z1, x2, y2, z2
  # it returns a distance
  def distance_between(x1, y1, z1, x2, y2, z2):
    distsquared = (x2-x1)*(x2-x1)+(y2-y1)*(y2-y1)+(z2-z1)*(z2-z1)
    dist = sqrt(distsquared)
    return dist
  end

  # this function takes a point, a unit vector, and a distance, and adds the distance to the point in the direction of the unit vector (3d space)
  # it returns a point as a list of coordinates
  def add_vectordistance_to_point(xi, yi, zi, uvx, uvy, uvz, delta):
    xf = xi + uvx * delta
    yf = yi + uvy * delta
    zf = zi + uvz * delta
    ret = [xf, yf, zf]
    return ret
  end

  # this function converts a heading (ccw radians from the positive x axis) into rxryrz to be put into a point p[]
  def convert_heading_to_axang(heading):
   axisxraw = -1 * sin(heading)
   axisyraw = cos(heading) + 1
   axiszraw = sin(heading)

   magnitude = sqrt(axisxraw*axisxraw + axisyraw*axisyraw + axiszraw*axiszraw)

   axisxunit = axisxraw / magnitude
   axisyunit = axisyraw / magnitude
   axiszunit = axiszraw / magnitude

   angle = acos( (cos(heading) - 1) / 2 )

   rxout = axisxunit * angle
   ryout = axisyunit * angle
   rzout = axiszunit * angle

   return [rxout, ryout, rzout]
  end

  $ 7 "path1≔analyze_touchpoints(p11,p12,p21,p22,p3)"
  global path1=analyze_touchpoints(p11,p12,p21,p22,p3)
  $ 8 "Call move_path_2"
  move_path_2()
end
